{attribute addProperty BoxType "EK1100-0000-0018"}
{attribute addProperty Id "Beckhoff_EL9xxxEK1122Beckhoff_EL9xxxEK1122_2D49AF05162A_0003_EL9110_0000_0016EL9110_CB6430E0405A_0004_EL9110_0000_0017EL9110_CB6430E0405A_0005_EL9110_0000_0018EL9110_CB6430E0405A_0006_EL9160_0000_0016EL9160_CB6430E0405A_0007_EL9210_0000_0016EL9210_F97BC8F0486A_0008_EL9210_0000_0017EL9210_F97BC8F0486A_0009_EL9210_0000_0018EL9210_F97BC8F0486A_0010_EL9210_0020_0016EL9210_F97BC8F0486A_0011_EL9210_0020_0017EL9210_F97BC8F0486A_0012_EL9210_0020_0018EL9210_F97BC8F0486A_0013_EL9221_4030_0018EL9221_0E81876614418A_0014_EL9221_5000_0018EL9221_0E81876614418A_0015_EL9221_5090_0018EL9221_0E81876614418A_0016_EL9221_6000_0018EL9221_0E81876614418A_0017_EL9221_6040_0018EL9221_0E81876614418A_0018_EL9221_9060_0018EL9221_0E81876614418A_0019_EL9221_9080_0018EL9221_0E81876614418A_0020_EL9222_4433_0018EL9222_39D75EBE19224A_0021_EL9222_5500_0018EL9222_39D75EBE19224A_0022_EL9222_6600_0018EL9222_39D75EBE19224A_0023_EL9222_6644_0018EL9222_39D75EBE19224A_0024_EL9222_9482_0018EL9222_39D75EBE19224A_0025_EL9222_9664_0018EL9222_39D75EBE19224A_0026_EL9227_4433_0018EL9227_9EBC899732040A_0027_EL9227_5500_0018EL9227_9EBC899732040A_0028_EL9227_6600_0018EL9227_9EBC899732040A_0029_EL9227_6644_0018EL9227_9EBC899732040A_0030_EL9227_9482_0018EL9227_9EBC899732040A_0031_EL9227_9664_0018EL9227_9EBC899732040A_0032_EL9260_0000_0016EL9260_F97BC8F0486A_0033_EL9410_0000_0016EL9410_D787878A486A_0034_EL9410_0000_0017EL9410_D787878A486A_0035_EL9505_0000_0016EL9505_A1085FEB486A_0036_EL9505_0000_0017EL9505_A1085FEB486A_0037_EL9505_0000_0018EL9505_A1085FEB486A_0038_EL9508_0000_0016EL9508_A1085FEB486A_0039_EL9508_0000_0017EL9508_A1085FEB486A_0040_EL9508_0000_0018EL9508_A1085FEB486A_0041_EL9510_0000_0016EL9510_A1085FEB486A_0042_EL9510_0000_0017EL9510_A1085FEB486A_0043_EL9510_0000_0018EL9510_A1085FEB486A_0044_EL9512_0000_0016EL9512_A1085FEB486A_0045_EL9512_0000_0017EL9512_A1085FEB486A_0046_EL9512_0000_0018EL9512_A1085FEB486A_0047_EL9515_0000_0016EL9515_A1085FEB486A_0048_EL9515_0000_0017EL9515_A1085FEB486A_0049_EL9515_0000_0018EL9515_A1085FEB486A_0050_EL9520_0000_0016EL9520_3B4447B6405A_0051_EL9520_0000_0017EL9520_3B4447B6405A_0052_EL9540_0010_0016EL9540_7D2BCDCD486A_0053_EL9550_0010_0016EL9550_E584A12F648A_0054_EL9560_0000_0016EL9560_A2048F02486A_0055_EL9560_0000_0017EL9560_A2048F02486A_0056_EL9560_0000_0018EL9560_A2048F02486A_0057_EL9576_0000_0016EL9576_4694F56721627A_0058_EL9576_0000_0017EL9576_37EDA20522428A_0059_EL9576_0000_0018EL9576_37EDA20522428A_0060_EL9576_0000_0019EL9576_A45E449923229A_0061_EL9576_0000_0020EL9576_57CA9E3622428A_0062_EL9576_0000_0021EL9576_57CA9E3622428A_0063_EL9576_0000_0022EL9576_B5DF83EF23229A_0086_EL9540_0010EL9540_7D2BCDCD486A_0088_EL9550_0010EL9550_E584A12F648"}
{attribute addProperty CRC "1772735843"}
{attribute addProperty SizeInBites "7432"}
{attribute addProperty SizeInBytes "929"}
TYPE Beckhoff_EL9xxx_69A9CD63 EXTENDS EK1100_179A0949 :
STRUCT
	{attribute addProperty Name "Beckhoff_EL9xxxEK1122"}
	Beckhoff_EL9xxxEK1122 : Beckhoff_EL9xxxEK1122_2D49AF05;
	{attribute addProperty Name "A_0003_EL9110_0000_0016"}
	A_0003_EL9110_0000_0016 : EL9110_CB6430E0;
	{attribute addProperty Name "A_0004_EL9110_0000_0017"}
	A_0004_EL9110_0000_0017 : EL9110_CB6430E0;
	{attribute addProperty Name "A_0005_EL9110_0000_0018"}
	A_0005_EL9110_0000_0018 : EL9110_CB6430E0;
	{attribute addProperty Name "A_0006_EL9160_0000_0016"}
	A_0006_EL9160_0000_0016 : EL9160_CB6430E0;
	{attribute addProperty Name "A_0007_EL9210_0000_0016"}
	A_0007_EL9210_0000_0016 : EL9210_F97BC8F0;
	{attribute addProperty Name "A_0008_EL9210_0000_0017"}
	A_0008_EL9210_0000_0017 : EL9210_F97BC8F0;
	{attribute addProperty Name "A_0009_EL9210_0000_0018"}
	A_0009_EL9210_0000_0018 : EL9210_F97BC8F0;
	{attribute addProperty Name "A_0010_EL9210_0020_0016"}
	A_0010_EL9210_0020_0016 : EL9210_F97BC8F0;
	{attribute addProperty Name "A_0011_EL9210_0020_0017"}
	A_0011_EL9210_0020_0017 : EL9210_F97BC8F0;
	{attribute addProperty Name "A_0012_EL9210_0020_0018"}
	A_0012_EL9210_0020_0018 : EL9210_F97BC8F0;
	{attribute addProperty Name "A_0013_EL9221_4030_0018"}
	A_0013_EL9221_4030_0018 : EL9221_0E818766;
	{attribute addProperty Name "A_0014_EL9221_5000_0018"}
	A_0014_EL9221_5000_0018 : EL9221_0E818766;
	{attribute addProperty Name "A_0015_EL9221_5090_0018"}
	A_0015_EL9221_5090_0018 : EL9221_0E818766;
	{attribute addProperty Name "A_0016_EL9221_6000_0018"}
	A_0016_EL9221_6000_0018 : EL9221_0E818766;
	{attribute addProperty Name "A_0017_EL9221_6040_0018"}
	A_0017_EL9221_6040_0018 : EL9221_0E818766;
	{attribute addProperty Name "A_0018_EL9221_9060_0018"}
	A_0018_EL9221_9060_0018 : EL9221_0E818766;
	{attribute addProperty Name "A_0019_EL9221_9080_0018"}
	A_0019_EL9221_9080_0018 : EL9221_0E818766;
	{attribute addProperty Name "A_0020_EL9222_4433_0018"}
	A_0020_EL9222_4433_0018 : EL9222_39D75EBE;
	{attribute addProperty Name "A_0021_EL9222_5500_0018"}
	A_0021_EL9222_5500_0018 : EL9222_39D75EBE;
	{attribute addProperty Name "A_0022_EL9222_6600_0018"}
	A_0022_EL9222_6600_0018 : EL9222_39D75EBE;
	{attribute addProperty Name "A_0023_EL9222_6644_0018"}
	A_0023_EL9222_6644_0018 : EL9222_39D75EBE;
	{attribute addProperty Name "A_0024_EL9222_9482_0018"}
	A_0024_EL9222_9482_0018 : EL9222_39D75EBE;
	{attribute addProperty Name "A_0025_EL9222_9664_0018"}
	A_0025_EL9222_9664_0018 : EL9222_39D75EBE;
	{attribute addProperty Name "A_0026_EL9227_4433_0018"}
	A_0026_EL9227_4433_0018 : EL9227_9EBC8997;
	{attribute addProperty Name "A_0027_EL9227_5500_0018"}
	A_0027_EL9227_5500_0018 : EL9227_9EBC8997;
	{attribute addProperty Name "A_0028_EL9227_6600_0018"}
	A_0028_EL9227_6600_0018 : EL9227_9EBC8997;
	{attribute addProperty Name "A_0029_EL9227_6644_0018"}
	A_0029_EL9227_6644_0018 : EL9227_9EBC8997;
	{attribute addProperty Name "A_0030_EL9227_9482_0018"}
	A_0030_EL9227_9482_0018 : EL9227_9EBC8997;
	{attribute addProperty Name "A_0031_EL9227_9664_0018"}
	A_0031_EL9227_9664_0018 : EL9227_9EBC8997;
	{attribute addProperty Name "A_0032_EL9260_0000_0016"}
	A_0032_EL9260_0000_0016 : EL9260_F97BC8F0;
	{attribute addProperty Name "A_0033_EL9410_0000_0016"}
	A_0033_EL9410_0000_0016 : EL9410_D787878A;
	{attribute addProperty Name "A_0034_EL9410_0000_0017"}
	A_0034_EL9410_0000_0017 : EL9410_D787878A;
	{attribute addProperty Name "A_0035_EL9505_0000_0016"}
	A_0035_EL9505_0000_0016 : EL9505_A1085FEB;
	{attribute addProperty Name "A_0036_EL9505_0000_0017"}
	A_0036_EL9505_0000_0017 : EL9505_A1085FEB;
	{attribute addProperty Name "A_0037_EL9505_0000_0018"}
	A_0037_EL9505_0000_0018 : EL9505_A1085FEB;
	{attribute addProperty Name "A_0038_EL9508_0000_0016"}
	A_0038_EL9508_0000_0016 : EL9508_A1085FEB;
	{attribute addProperty Name "A_0039_EL9508_0000_0017"}
	A_0039_EL9508_0000_0017 : EL9508_A1085FEB;
	{attribute addProperty Name "A_0040_EL9508_0000_0018"}
	A_0040_EL9508_0000_0018 : EL9508_A1085FEB;
	{attribute addProperty Name "A_0041_EL9510_0000_0016"}
	A_0041_EL9510_0000_0016 : EL9510_A1085FEB;
	{attribute addProperty Name "A_0042_EL9510_0000_0017"}
	A_0042_EL9510_0000_0017 : EL9510_A1085FEB;
	{attribute addProperty Name "A_0043_EL9510_0000_0018"}
	A_0043_EL9510_0000_0018 : EL9510_A1085FEB;
	{attribute addProperty Name "A_0044_EL9512_0000_0016"}
	A_0044_EL9512_0000_0016 : EL9512_A1085FEB;
	{attribute addProperty Name "A_0045_EL9512_0000_0017"}
	A_0045_EL9512_0000_0017 : EL9512_A1085FEB;
	{attribute addProperty Name "A_0046_EL9512_0000_0018"}
	A_0046_EL9512_0000_0018 : EL9512_A1085FEB;
	{attribute addProperty Name "A_0047_EL9515_0000_0016"}
	A_0047_EL9515_0000_0016 : EL9515_A1085FEB;
	{attribute addProperty Name "A_0048_EL9515_0000_0017"}
	A_0048_EL9515_0000_0017 : EL9515_A1085FEB;
	{attribute addProperty Name "A_0049_EL9515_0000_0018"}
	A_0049_EL9515_0000_0018 : EL9515_A1085FEB;
	{attribute addProperty Name "A_0050_EL9520_0000_0016"}
	A_0050_EL9520_0000_0016 : EL9520_3B4447B6;
	{attribute addProperty Name "A_0051_EL9520_0000_0017"}
	A_0051_EL9520_0000_0017 : EL9520_3B4447B6;
	{attribute addProperty Name "A_0052_EL9540_0010_0016"}
	A_0052_EL9540_0010_0016 : EL9540_7D2BCDCD;
	{attribute addProperty Name "A_0053_EL9550_0010_0016"}
	A_0053_EL9550_0010_0016 : EL9550_E584A12F;
	{attribute addProperty Name "A_0054_EL9560_0000_0016"}
	A_0054_EL9560_0000_0016 : EL9560_A2048F02;
	{attribute addProperty Name "A_0055_EL9560_0000_0017"}
	A_0055_EL9560_0000_0017 : EL9560_A2048F02;
	{attribute addProperty Name "A_0056_EL9560_0000_0018"}
	A_0056_EL9560_0000_0018 : EL9560_A2048F02;
	{attribute addProperty Name "A_0057_EL9576_0000_0016"}
	A_0057_EL9576_0000_0016 : EL9576_4694F567;
	{attribute addProperty Name "A_0058_EL9576_0000_0017"}
	A_0058_EL9576_0000_0017 : EL9576_37EDA205;
	{attribute addProperty Name "A_0059_EL9576_0000_0018"}
	A_0059_EL9576_0000_0018 : EL9576_37EDA205;
	{attribute addProperty Name "A_0060_EL9576_0000_0019"}
	A_0060_EL9576_0000_0019 : EL9576_A45E4499;
	{attribute addProperty Name "A_0061_EL9576_0000_0020"}
	A_0061_EL9576_0000_0020 : EL9576_57CA9E36;
	{attribute addProperty Name "A_0062_EL9576_0000_0021"}
	A_0062_EL9576_0000_0021 : EL9576_57CA9E36;
	{attribute addProperty Name "A_0063_EL9576_0000_0022"}
	A_0063_EL9576_0000_0022 : EL9576_B5DF83EF;
	{attribute addProperty Name "A_0086_EL9540_0010"}
	A_0086_EL9540_0010 : EL9540_7D2BCDCD;
	{attribute addProperty Name "A_0088_EL9550_0010"}
	A_0088_EL9550_0010 : EL9550_E584A12F;
END_STRUCT
END_TYPE

(* stored: Version 1.2.0.0, ProductVersion 3.1.4024.9
   DUT Beckhoff_EL9xxx_69A9CD63: Id {7a460b07-d62c-473b-9727-1965856bbcb1} *)
